Staubli VAL3: getSize.pgx

public program getSize(num& nSize[])
begin
  nSize=size(saveTool:gun)
end
